{attribute 'qualified_only'}
{attribute 'strict'}
TYPE States :
(
	Reset := 0,
	Init,
	Enable,
	bLocal,
	MoveType,
	Error,
	Absolute,
	Relative,
	Velocity,
	Stop
);
END_TYPE

(* stored: Version 1.1.0.1, ProductVersion 3.1.4024.9
   DUT States: Id {d04e3668-c687-4493-acb3-0bc833cea6d9} *)
